SPLINE
SPL {X  -158.679, Y  +692.020, Z    +0.000, E1   -14.212, E3 +179990.334}
SPL {X  -159.747, Y  +680.500, Z    +0.000, E1    -7.378, E3 +179998.711}
SPL {X  -160.000, Y  +671.618, Z    +0.000, E1    -1.592, E3 +180002.326}
SPL {X  -160.000, Y  +666.041, Z    +0.000, E1    +2.615, E3 +180004.292}
SPL {X  -160.000, Y  +661.396, Z    +0.000, E1    +6.484, E3 +180005.965}
SPL {X  -160.000, Y  +653.532, Z    +0.000, E1   +13.136, E3 +180010.086}
SPL {X  -160.000, Y  +631.927, Z    +0.000, E1   +26.832, E3 +180032.852}
SPL {X  -160.000, Y  +610.736, Z    +0.000, E1   +32.114, E3 +180075.522}
SPL {X  -160.000, Y  +605.907, Z    +0.000, E1   +32.114, E3 +180091.870}
SPL {X  -160.000, Y  +601.221, Z    +0.000, E1   +32.108, E3 +180107.737}
SPL {X  -160.000, Y  +596.433, Z    +0.000, E1   +32.120, E3 +180123.920}
SPL {X  -160.000, Y  +592.025, Z    +0.000, E1   +32.104, E3 +180138.844}
SPL {X  -160.000, Y  +587.734, Z    +0.000, E1   +32.110, E3 +180153.364}
SPL {X  -160.000, Y  +583.150, Z    +0.000, E1   +32.111, E3 +180168.892}
SPL {X  -160.000, Y  +579.063, Z    +0.000, E1   +32.085, E3 +180182.793}
SPL {X  -160.000, Y  +574.897, Z    +0.000, E1   +32.110, E3 +180196.845}
SPL {X  -160.000, Y  +570.471, Z    +0.000, E1   +32.093, E3 +180211.859}
SPL {X  -160.000, Y  +566.667, Z    +0.000, E1   +32.086, E3 +180224.773}
SPL {X  -160.000, Y  +562.434, Z    +0.000, E1   +32.097, E3 +180239.083}
SPL {X  -160.000, Y  +557.710, Z    +0.000, E1   +32.104, E3 +180255.066}
SPL {X  -160.000, Y  +553.479, Z    +0.000, E1   +32.081, E3 +180269.436}
SPL {X  -160.000, Y  +547.489, Z    +0.000, E1   +32.181, E3 +180289.554}
SPL {X  -160.000, Y  +541.554, Z    +0.000, E1   +32.092, E3 +180309.791}
SPL {X  -160.000, Y  +537.332, Z    +0.000, E1   +32.092, E3 +180324.089}
SPL {X  -160.000, Y  +533.113, Z    +0.000, E1   +32.090, E3 +180338.385}
SPL {X  -160.000, Y  +528.875, Z    +0.000, E1   +32.090, E3 +180352.729}
SPL {X  -160.000, Y  +524.453, Z    +0.000, E1   +32.104, E3 +180367.653}
SPL {X  -160.000, Y  +520.037, Z    +0.000, E1   +32.096, E3 +180382.595}
SPL {X  -160.000, Y  +514.030, Z    +0.000, E1   +32.182, E3 +180402.791}
SPL {X  -160.000, Y  +508.131, Z    +0.000, E1   +32.099, E3 +180422.895}
SPL {X  -160.000, Y  +504.077, Z    +0.000, E1   +32.094, E3 +180436.618}
SPL {X  -160.000, Y  +494.657, Z    +0.000, E1   +34.509, E3 +180451.481}
SPL {X  -160.000, Y  +491.565, Z    +0.000, E1   +33.823, E3 +180465.388}
SPL {X  -160.000, Y  +489.317, Z    +0.000, E1   +32.894, E3 +180478.733}
SPL {X  -160.000, Y  +486.958, Z    +0.000, E1   +31.703, E3 +180494.505}
SPL {X  -160.000, Y  +484.144, Z    +0.000, E1   +30.999, E3 +180508.928}
SPL {X  -160.000, Y  +479.156, Z    +0.000, E1   +31.035, E3 +180526.494}
SPL {X  -160.000, Y  +474.045, Z    +0.000, E1   +31.015, E3 +180544.585}
SPL {X  -160.000, Y  +468.999, Z    +0.000, E1   +31.021, E3 +180562.410}
SPL {X  -160.000, Y  +464.107, Z    +0.000, E1   +31.012, E3 +180579.710}
SPL {X  -160.000, Y  +459.262, Z    +0.000, E1   +31.016, E3 +180596.817}
SPL {X  -160.000, Y  +454.119, Z    +0.000, E1   +31.026, E3 +180614.967}
SPL {X  -160.000, Y  +448.874, Z    +0.000, E1   +31.019, E3 +180633.523}
SPL {X  -160.000, Y  +443.892, Z    +0.000, E1   +31.019, E3 +180651.111}
SPL {X  -160.000, Y  +438.782, Z    +0.000, E1   +31.022, E3 +180669.185}
SPL {X  -160.000, Y  +433.722, Z    +0.000, E1   +31.007, E3 +180687.129}
SPL {X  -160.000, Y  +428.980, Z    +0.000, E1   +31.004, E3 +180703.886}
SPL {X  -160.000, Y  +424.339, Z    +0.000, E1   +31.006, E3 +180720.261}
SPL {X  -160.000, Y  +419.231, Z    +0.000, E1   +31.030, E3 +180738.254}
SPL {X  -160.000, Y  +414.179, Z    +0.000, E1   +31.008, E3 +180756.151}
SPL {X  -160.000, Y  +409.416, Z    +0.000, E1   +31.023, E3 +180772.935}
SPL {X  -160.000, Y  +403.994, Z    +0.000, E1   +31.033, E3 +180792.090}
SPL {X  -160.000, Y  +399.052, Z    +0.000, E1   +31.010, E3 +180809.558}
SPL {X  -160.000, Y  +394.012, Z    +0.000, E1   +31.036, E3 +180827.347}
SPL {X  -159.999, Y  +388.376, Z    +0.000, E1   +31.028, E3 +180847.277}
SPL {X  -159.897, Y  +383.070, Z    +0.000, E1   +31.010, E3 +180866.115}
SPL {X  -159.656, Y  +378.313, Z    +0.000, E1   +30.961, E3 +180883.207}
SPL {X  -159.237, Y  +373.190, Z    +0.000, E1   +30.917, E3 +180901.707}
SPL {X  -158.628, Y  +367.891, Z    +0.000, E1   +30.812, E3 +180921.093}
SPL {X  -157.915, Y  +363.053, Z    +0.000, E1   +30.689, E3 +180938.960}
SPL {X  -157.216, Y  +359.084, Z    +0.000, E1   +30.550, E3 +180953.762}
SPL {X  -156.248, Y  +354.355, Z    +0.000, E1   +30.460, E3 +180971.375}
SPL {X  -155.629, Y  +351.657, Z    +0.000, E1   +25.972, E3 +181017.803}
ENDSPLINE

SPLINE
SPL {X  -156.240, Y  +354.319, Z    +0.000, E1   +23.538, E3 +181030.411}
SPL {X  -159.137, Y  +372.201, Z    +0.000, E1   +12.017, E3 +181060.248}
SPL {X  -159.858, Y  +382.069, Z    +0.000, E1    +5.945, E3 +181066.766}
SPL {X  -160.000, Y  +389.339, Z    +0.000, E1    +1.101, E3 +181069.928}
SPL {X  -160.000, Y  +395.749, Z    +0.000, E1    -3.722, E3 +181072.533}
SPL {X  -160.000, Y  +403.128, Z    +0.000, E1    -9.899, E3 +181075.837}
SPL {X  -160.000, Y  +411.609, Z    +0.000, E1   -16.851, E3 +181081.158}
SPL {X  -160.000, Y  +429.715, Z    +0.000, E1   -27.376, E3 +181100.522}
SPL {X  -160.000, Y  +449.791, Z    +0.000, E1   -32.145, E3 +181141.759}
SPL {X  -160.000, Y  +454.903, Z    +0.000, E1   -32.134, E3 +181159.063}
SPL {X  -160.000, Y  +460.041, Z    +0.000, E1   -32.144, E3 +181176.416}
SPL {X  -160.000, Y  +465.466, Z    +0.000, E1   -32.152, E3 +181194.734}
SPL {X  -160.000, Y  +471.112, Z    +0.000, E1   -32.154, E3 +181213.822}
SPL {X  -160.000, Y  +476.735, Z    +0.000, E1   -32.156, E3 +181232.813}
SPL {X  -160.000, Y  +482.675, Z    +0.000, E1   -32.169, E3 +181252.862}
SPL {X  -160.000, Y  +488.008, Z    +0.000, E1   -32.144, E3 +181270.909}
SPL {X  -160.000, Y  +493.245, Z    +0.000, E1   -32.159, E3 +181288.617}
SPL {X  -160.000, Y  +498.210, Z    +0.000, E1   -32.128, E3 +181305.452}
SPL {X  -160.000, Y  +503.407, Z    +0.000, E1   -32.165, E3 +181322.955}
SPL {X  -160.000, Y  +509.142, Z    +0.000, E1   -32.157, E3 +181342.351}
SPL {X  -160.000, Y  +514.696, Z    +0.000, E1   -32.156, E3 +181361.131}
SPL {X  -160.000, Y  +520.339, Z    +0.000, E1   -32.159, E3 +181380.204}
SPL {X  -160.000, Y  +525.825, Z    +0.000, E1   -32.148, E3 +181398.767}
SPL {X  -160.000, Y  +530.379, Z    +0.000, E1   -32.130, E3 +181414.195}
SPL {X  -160.000, Y  +535.020, Z    +0.000, E1   -32.146, E3 +181429.841}
SPL {X  -160.000, Y  +540.303, Z    +0.000, E1   -32.158, E3 +181447.667}
SPL {X  -160.000, Y  +545.740, Z    +0.000, E1   -32.155, E3 +181466.059}
SPL {X  -160.000, Y  +550.807, Z    +0.000, E1   -32.147, E3 +181483.182}
SPL {X  -160.000, Y  +555.841, Z    +0.000, E1   -32.148, E3 +181500.221}
SPL {X  -160.000, Y  +561.018, Z    +0.000, E1   -32.143, E3 +181517.750}
SPL {X  -160.000, Y  +566.466, Z    +0.000, E1   -32.153, E3 +181536.168}
SPL {X  -160.000, Y  +571.733, Z    +0.000, E1   -32.135, E3 +181554.005}
SPL {X  -160.000, Y  +576.943, Z    +0.000, E1   -32.148, E3 +181571.602}
SPL {X  -160.000, Y  +582.183, Z    +0.000, E1   -32.140, E3 +181589.327}
SPL {X  -160.000, Y  +587.036, Z    +0.000, E1   -32.141, E3 +181605.697}
SPL {X  -160.000, Y  +591.785, Z    +0.000, E1   -32.144, E3 +181621.721}
SPL {X  -160.000, Y  +596.962, Z    +0.000, E1   -32.161, E3 +181639.208}
SPL {X  -160.000, Y  +601.800, Z    +0.000, E1   -32.134, E3 +181655.605}
SPL {X  -160.000, Y  +606.611, Z    +0.000, E1   -32.156, E3 +181671.819}
SPL {X  -160.000, Y  +611.219, Z    +0.000, E1   -32.131, E3 +181687.433}
SPL {X  -160.000, Y  +616.331, Z    +0.000, E1   -32.174, E3 +181704.630}
SPL {X  -160.000, Y  +621.751, Z    +0.000, E1   -32.150, E3 +181722.973}
SPL {X  -160.000, Y  +626.312, Z    +0.000, E1   -32.145, E3 +181738.379}
SPL {X  -160.000, Y  +630.971, Z    +0.000, E1   -32.155, E3 +181754.107}
SPL {X  -160.000, Y  +635.550, Z    +0.000, E1   -32.137, E3 +181769.633}
SPL {X  -160.000, Y  +640.419, Z    +0.000, E1   -32.158, E3 +181786.071}
SPL {X  -160.000, Y  +645.749, Z    +0.000, E1   -32.151, E3 +181804.096}
SPL {X  -160.000, Y  +650.662, Z    +0.000, E1   -32.150, E3 +181820.667}
SPL {X  -160.000, Y  +655.372, Z    +0.000, E1   -32.145, E3 +181836.614}
SPL {X  -160.000, Y  +660.593, Z    +0.000, E1   -32.163, E3 +181854.232}
SPL {X  -160.000, Y  +665.836, Z    +0.000, E1   -32.154, E3 +181871.949}
SPL {X  -160.000, Y  +670.613, Z    +0.000, E1   -32.138, E3 +181888.159}
SPL {X  -159.954, Y  +675.336, Z    +0.000, E1   -32.135, E3 +181904.167}
SPL {X  -159.758, Y  +680.302, Z    +0.000, E1   -32.108, E3 +181921.182}
SPL {X  -159.416, Y  +685.158, Z    +0.000, E1   -32.039, E3 +181937.993}
SPL {X  -158.953, Y  +689.772, Z    +0.000, E1   -31.965, E3 +181954.092}
SPL {X  -158.363, Y  +694.328, Z    +0.000, E1   -31.871, E3 +181970.105}
SPL {X  -157.606, Y  +699.074, Z    +0.000, E1   -31.756, E3 +181986.948}
SPL {X  -156.791, Y  +703.384, Z    +0.000, E1   -31.607, E3 +182002.399}
SPL {X  -155.792, Y  +707.952, Z    +0.000, E1   -31.465, E3 +182018.845}
SPL {X  -155.149, Y  +710.598, Z    +0.000, E1   -26.183, E3 +182074.305}
ENDSPLINE

SPLINE
SPL {X  -158.679, Y  +692.020, Z    +0.000, E1   -14.212, E3 +182107.981}
SPL {X  -159.747, Y  +680.500, Z    +0.000, E1    -7.378, E3 +182116.359}
SPL {X  -160.000, Y  +671.618, Z    +0.000, E1    -1.592, E3 +182119.973}
SPL {X  -160.000, Y  +666.041, Z    +0.000, E1    +2.615, E3 +182121.940}
SPL {X  -160.000, Y  +661.396, Z    +0.000, E1    +6.484, E3 +182123.613}
SPL {X  -160.000, Y  +653.532, Z    +0.000, E1   +13.136, E3 +182127.733}
SPL {X  -160.000, Y  +631.927, Z    +0.000, E1   +26.832, E3 +182150.500}
SPL {X  -160.000, Y  +610.736, Z    +0.000, E1   +32.114, E3 +182193.169}
SPL {X  -160.000, Y  +605.907, Z    +0.000, E1   +32.114, E3 +182209.517}
SPL {X  -160.000, Y  +601.221, Z    +0.000, E1   +32.108, E3 +182225.385}
SPL {X  -160.000, Y  +596.433, Z    +0.000, E1   +32.120, E3 +182241.567}
SPL {X  -160.000, Y  +592.025, Z    +0.000, E1   +32.104, E3 +182256.491}
SPL {X  -160.000, Y  +587.734, Z    +0.000, E1   +32.110, E3 +182271.012}
SPL {X  -160.000, Y  +583.150, Z    +0.000, E1   +32.111, E3 +182286.539}
SPL {X  -160.000, Y  +579.063, Z    +0.000, E1   +32.085, E3 +182300.441}
SPL {X  -160.000, Y  +574.897, Z    +0.000, E1   +32.110, E3 +182314.492}
SPL {X  -160.000, Y  +570.471, Z    +0.000, E1   +32.093, E3 +182329.506}
SPL {X  -160.000, Y  +566.667, Z    +0.000, E1   +32.086, E3 +182342.421}
SPL {X  -160.000, Y  +562.434, Z    +0.000, E1   +32.097, E3 +182356.730}
SPL {X  -160.000, Y  +557.710, Z    +0.000, E1   +32.104, E3 +182372.714}
SPL {X  -160.000, Y  +553.479, Z    +0.000, E1   +32.081, E3 +182387.083}
SPL {X  -160.000, Y  +547.489, Z    +0.000, E1   +32.181, E3 +182407.202}
SPL {X  -160.000, Y  +541.554, Z    +0.000, E1   +32.092, E3 +182427.439}
SPL {X  -160.000, Y  +537.332, Z    +0.000, E1   +32.092, E3 +182441.736}
SPL {X  -160.000, Y  +533.113, Z    +0.000, E1   +32.090, E3 +182456.033}
SPL {X  -160.000, Y  +528.875, Z    +0.000, E1   +32.090, E3 +182470.376}
SPL {X  -160.000, Y  +524.453, Z    +0.000, E1   +32.104, E3 +182485.300}
SPL {X  -160.000, Y  +520.037, Z    +0.000, E1   +32.096, E3 +182500.242}
SPL {X  -160.000, Y  +514.030, Z    +0.000, E1   +32.182, E3 +182520.438}
SPL {X  -160.000, Y  +508.131, Z    +0.000, E1   +32.099, E3 +182540.542}
SPL {X  -160.000, Y  +504.077, Z    +0.000, E1   +32.094, E3 +182554.265}
SPL {X  -160.000, Y  +494.657, Z    +0.000, E1   +34.509, E3 +182569.128}
SPL {X  -160.000, Y  +491.565, Z    +0.000, E1   +33.823, E3 +182583.036}
SPL {X  -160.000, Y  +489.317, Z    +0.000, E1   +32.894, E3 +182596.380}
SPL {X  -160.000, Y  +486.958, Z    +0.000, E1   +31.703, E3 +182612.152}
ENDSPLINE

HALT
END
